FUNCTION_BLOCK FB_3_VerificarPale_SFC
VAR_INPUT
	
	//  SFC-Flags
	SFCPause: BOOL;
	SFCReset: BOOL;

	// Indicadores de sincronización
	Ack: BOOL := TRUE;
	Execute: BOOL;
	
	// Entradas
	VerificadorAbajo: BOOL;
	VerificadorArriba: BOOL;
	DesplazadorDetras: BOOL;
	TpoVerificador: TIME;
	TpoDesplazador: TIME;
	TpoRechazador: TIME;
	
END_VAR
VAR_OUTPUT
	
	// Indicadores de sincronización
	Ready: BOOL;	
	Done: BOOL;
	DoneIncorrecto: BOOL;
	// Salidas
	VerificadorBaja: BOOL;
	DesplazadorAdelante: BOOL;
	RechazadorAdelante: BOOL;
	
END_VAR

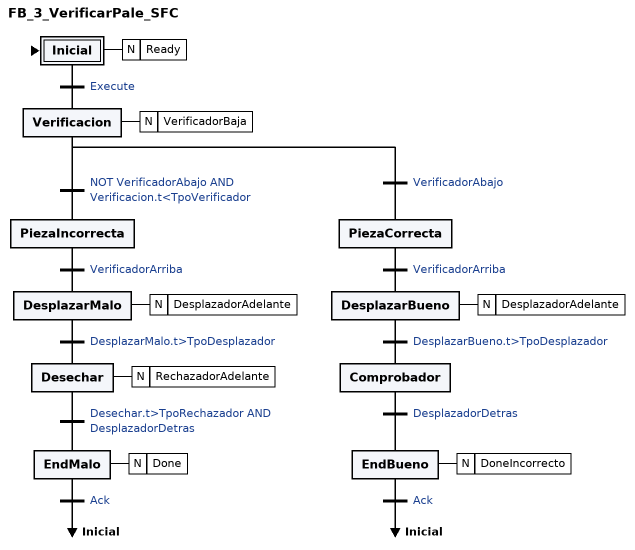
INITIAL_STEP Inicial:
    Ready(N);
END_STEP
TRANSITION FROM Inicial TO Verificacion
    := Execute;
END_TRANSITION
STEP Verificacion:
    VerificadorBaja(N);
END_STEP
TRANSITION FROM Verificacion TO PiezaIncorrecta
    := NOT VerificadorAbajo AND Verificacion.t<TpoVerificador;
END_TRANSITION
STEP PiezaIncorrecta:
END_STEP
TRANSITION FROM PiezaIncorrecta TO DesplazarMalo
    := VerificadorArriba;
END_TRANSITION
STEP DesplazarMalo:
    DesplazadorAdelante(N);
END_STEP
TRANSITION FROM DesplazarMalo TO Desechar
    := DesplazarMalo.t>TpoDesplazador;
END_TRANSITION
STEP Desechar:
    RechazadorAdelante(N);
END_STEP
TRANSITION FROM Desechar TO EndMalo
    := Desechar.t>TpoRechazador AND DesplazadorDetras;
END_TRANSITION
STEP EndMalo:
    Done(N);
END_STEP
TRANSITION FROM EndMalo TO Inicial
    := Ack;
END_TRANSITION
TRANSITION FROM Verificacion TO PiezaCorrecta
    := VerificadorAbajo;
END_TRANSITION
STEP PiezaCorrecta:
END_STEP
TRANSITION FROM PiezaCorrecta TO DesplazarBueno
    := VerificadorArriba;
END_TRANSITION
STEP DesplazarBueno:
    DesplazadorAdelante(N);
END_STEP
TRANSITION FROM DesplazarBueno TO Comprobador
    := DesplazarBueno.t>TpoDesplazador;
END_TRANSITION
STEP Comprobador:
END_STEP
TRANSITION FROM Comprobador TO EndBueno
    := DesplazadorDetras;
END_TRANSITION
STEP EndBueno:
    DoneIncorrecto(N);
END_STEP
TRANSITION FROM EndBueno TO Inicial
    := Ack;
END_TRANSITION

END_FUNCTION_BLOCK

(* stored: Version 1.1.0.1, ProductVersion 3.1.4024.12
   POU FB_3_VerificarPale_SFC: Id {b8ef243d-9616-4600-b196-4c2d11b3d533}, SpecialFunc None *)
